Staubli VAL3: login.pgx

public program login(sio& x_skSocketName[], string user_, string password_, num& handle_[], bool& result_[])
  local string strMsg
begin
  // login to camera via TCP/IP port 1023
  // x_skSocketName   : CS8 client socket with
  //                  IP address of camera
  //                  Port = 1023
  //                  Time Out = 0
  //                  End of line Char = 13
  //                  Nagle = On
  // user_     : user name
  // password_ : password for user user_
  // handle_   : returns a handle to camera for further operations
  // result_   : returns true if login succeeded
  //
  if bDebug
    putln("cognex login")
  endIf
  errorCode[handle_]=1
  nCommand[handle_]=coLO
  nHandleCount=nHandleCount+1
  handle_=nHandleCount
  sioLink(sSocket[handle_],x_skSocketName)
  // read welcome string
  call readSocket(handle_,strMsg,result_)
  // send user name
  call readLogin(handle_,strMsg,result_)
  call writeSocket(handle_,user_)
  // send password
  call readLogin(handle_,strMsg,result_)
  call writeSocket(handle_,password_)
  //
  // read login result
  call readSocket(handle_,strMsg,result_)
  result_=find(strMsg,"User Logged In")!=-1
  if !result_
    errorCode[handle_]=-1
    nHandleCount=nHandleCount-1
  else
  endIf
  if bDebug and !result_
    putln("login: login failed")
  endIf
end
